SUBAPPLICATION Funk_IXA_TO_DataPanel_MI_QXA (* Funk_IXA auf DataPanel_MI_QXA (generisch), adapter-basiert *)
  (* Standard: 61499-2 *)
  (* Version 1.0, 2026-09-09, Franz Höpfinger, Meisterschulen am Ostbahnhof, Ausgelagert aus Uebung_003b2_sub_AX (Uebung_003b3_sub_AX war ein exaktes Duplikat davon - entfernt, beide Parents zeigen jetzt hierher). *)
  PACKAGE MyLib::sys;
  IMPORT DataPanel::io::MI::DQ::DataPanel_MI_DO_S;
  IMPORT DataPanel::io::MI::const::MI;
  IMPORT Funk::io::DI::Funk_DI;
  IMPORT Funk::io::DI::Funk_DI_S;
  IMPORT DataPanel::io::MI::DQ::DataPanel_MI_DO::Invalid;
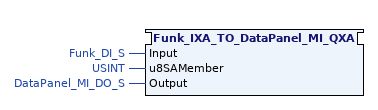
  VAR_INPUT
    Input : Funk::io::DI::Funk_DI_S := Funk_DI::Invalid; (* Identify the Input DigitalInput_Key_01 etc.. *)
    u8SAMember : USINT := MI::MI_00; (* Node SA 224..239 *)
    Output : DataPanel::io::MI::DQ::DataPanel_MI_DO_S := Invalid; (* Identify the Output DigitalOutput_1A..8B and Input_Power_Port_5..8 *)
  END_VAR
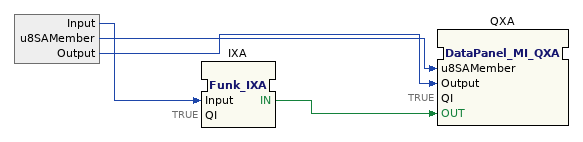
  FBS
    QXA : DataPanel::io::MI::DQ::DataPanel_MI_QXA(QI := TRUE);
    IXA : Funk::io::DI::Funk_IXA(QI := TRUE);
  END_FBS
  DATA_CONNECTIONS
    Input TO IXA.Input;
    u8SAMember TO QXA.u8SAMember;
    Output TO QXA.Output;
  END_CONNECTIONS
  ADAPTER_CONNECTIONS
    IXA.IN TO QXA.OUT;
  END_CONNECTIONS
END_SUBAPPLICATION
